// LS Electric XG5000 project: cobot_conveyor
// PLC LSPLC

PROGRAM InverterCom (task: 스캔 프로그램)

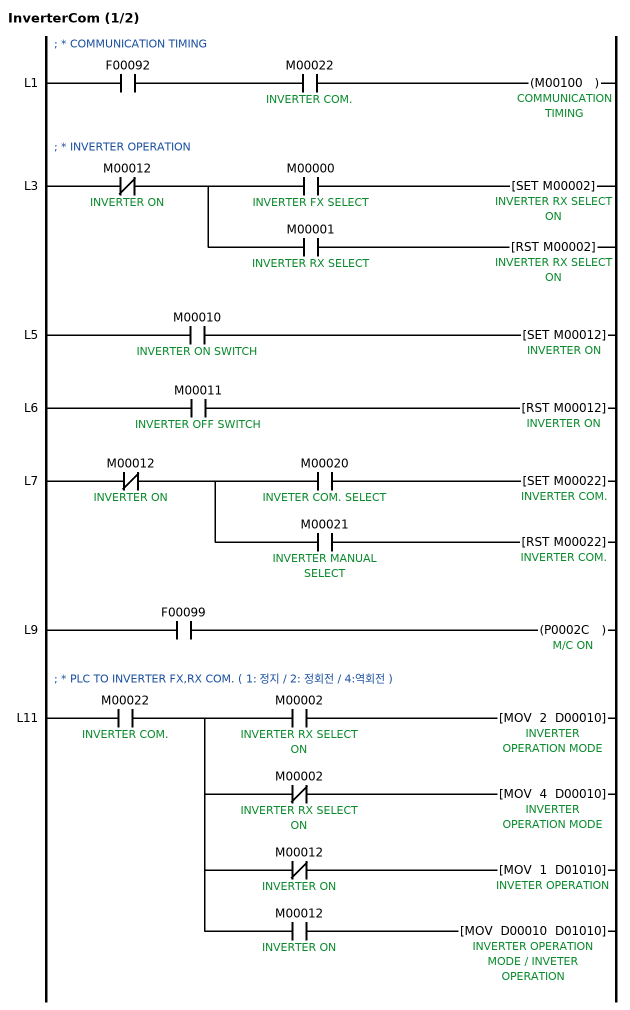
// * COMMUNICATION TIMING
; L1
LOAD      F00092
AND       M00022	// INVERTER COM.
OUT       M00100	// COMMUNICATION TIMING
// * INVERTER OPERATION
; L3
LOAD NOT  M00012	// INVERTER ON
MPUSH
AND       M00000	// INVERTER FX SELECT
SET       M00002	// INVERTER RX SELECT ON
MPOP
AND       M00001	// INVERTER RX SELECT
RST       M00002	// INVERTER RX SELECT ON
; L5
LOAD      M00010	// INVERTER ON SWITCH
SET       M00012	// INVERTER ON
; L6
LOAD      M00011	// INVERTER OFF SWITCH
RST       M00012	// INVERTER ON
; L7
LOAD NOT  M00012	// INVERTER ON
MPUSH
AND       M00020	// INVETER COM. SELECT
SET       M00022	// INVERTER COM.
MPOP
AND       M00021	// INVERTER MANUAL SELECT
RST       M00022	// INVERTER COM.
; L9
LOAD      F00099
OUT       P0002C	// M/C ON
// * PLC TO INVERTER FX,RX COM. ( 1: 정지 / 2: 정회전 / 4:역회전 )
; L11
LOAD      M00022	// INVERTER COM.
MPUSH
AND       M00002	// INVERTER RX SELECT ON
MOV       2 D00010	// INVERTER OPERATION MODE
MLOAD
AND NOT   M00002	// INVERTER RX SELECT ON
MOV       4 D00010	// INVERTER OPERATION MODE
MLOAD
AND NOT   M00012	// INVERTER ON
MOV       1 D01010	// INVETER OPERATION
MPOP
AND       M00012	// INVERTER ON
MOV       D00010 D01010	// INVERTER OPERATION MODE / INVETER OPERATION

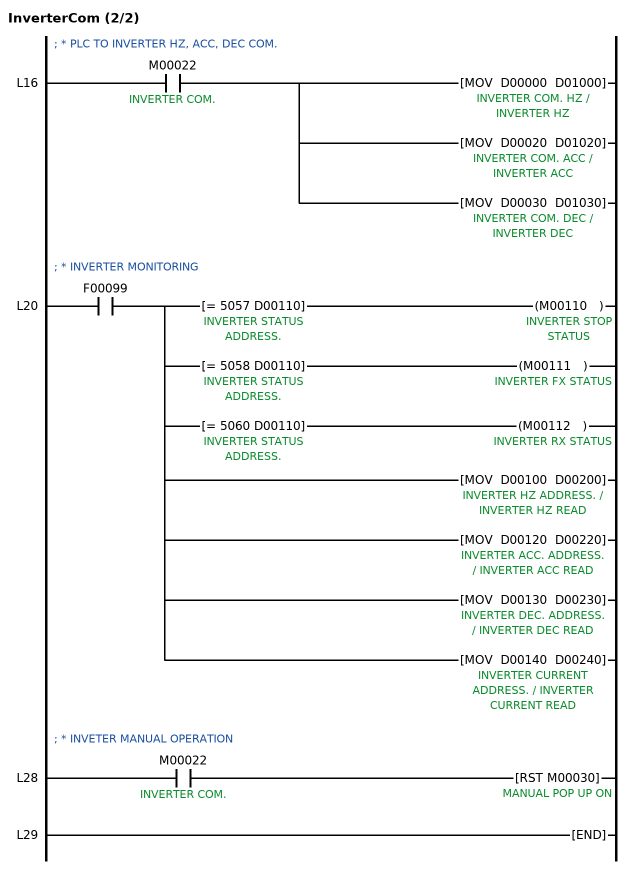
// * PLC TO INVERTER HZ, ACC, DEC COM.
; L16
LOAD      M00022	// INVERTER COM.
MOV       D00000 D01000	// INVERTER COM. HZ / INVERTER HZ
MOV       D00020 D01020	// INVERTER COM. ACC / INVERTER ACC
MOV       D00030 D01030	// INVERTER COM. DEC / INVERTER DEC
// * INVERTER MONITORING
; L20
LOAD      F00099
MPUSH
AND=      5057 D00110	// INVERTER STATUS ADDRESS.
OUT       M00110	// INVERTER STOP STATUS
MLOAD
AND=      5058 D00110	// INVERTER STATUS ADDRESS.
OUT       M00111	// INVERTER FX STATUS
MLOAD
AND=      5060 D00110	// INVERTER STATUS ADDRESS.
OUT       M00112	// INVERTER RX STATUS
MPOP
MOV       D00100 D00200	// INVERTER HZ ADDRESS. / INVERTER HZ READ
MOV       D00120 D00220	// INVERTER ACC. ADDRESS. / INVERTER ACC READ
MOV       D00130 D00230	// INVERTER DEC. ADDRESS. / INVERTER DEC READ
MOV       D00140 D00240	// INVERTER CURRENT ADDRESS. / INVERTER CURRENT READ
// * INVETER MANUAL OPERATION
; L28
LOAD      M00022	// INVERTER COM.
RST       M00030	// MANUAL POP UP ON
; L29
END

PROGRAM CountTimer (task: 스캔 프로그램)

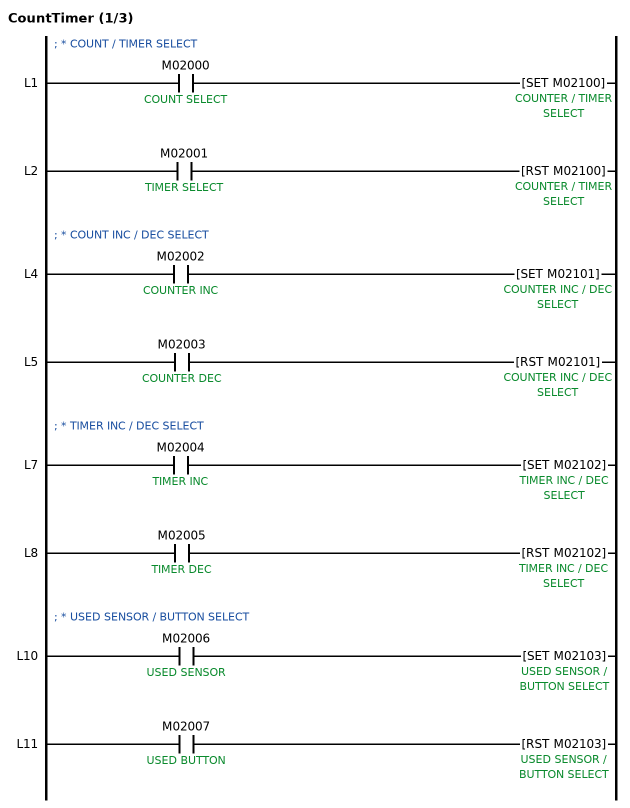
// * COUNT / TIMER SELECT
; L1
LOAD      M02000	// COUNT SELECT
SET       M02100	// COUNTER / TIMER SELECT
; L2
LOAD      M02001	// TIMER SELECT
RST       M02100	// COUNTER / TIMER SELECT
// * COUNT INC / DEC SELECT
; L4
LOAD      M02002	// COUNTER INC
SET       M02101	// COUNTER INC / DEC SELECT
; L5
LOAD      M02003	// COUNTER DEC
RST       M02101	// COUNTER INC / DEC SELECT
// * TIMER INC / DEC SELECT
; L7
LOAD      M02004	// TIMER INC
SET       M02102	// TIMER INC / DEC SELECT
; L8
LOAD      M02005	// TIMER DEC
RST       M02102	// TIMER INC / DEC SELECT
// * USED SENSOR / BUTTON SELECT
; L10
LOAD      M02006	// USED SENSOR
SET       M02103	// USED SENSOR / BUTTON SELECT
; L11
LOAD      M02007	// USED BUTTON
RST       M02103	// USED SENSOR / BUTTON SELECT

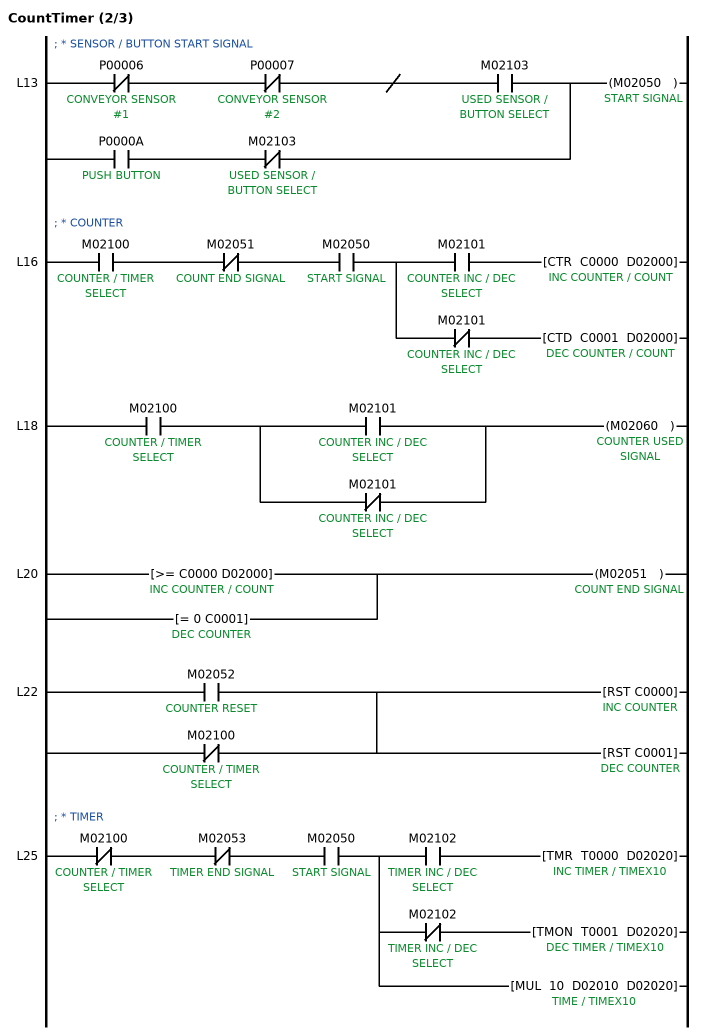
// * SENSOR / BUTTON START SIGNAL
; L13
LOAD NOT  P00006	// CONVEYOR SENSOR #1
AND NOT   P00007	// CONVEYOR SENSOR #2
NOT
AND       M02103	// USED SENSOR / BUTTON SELECT
LOAD      P0000A	// PUSH BUTTON
AND NOT   M02103	// USED SENSOR / BUTTON SELECT
OR LOAD
OUT       M02050	// START SIGNAL
// * COUNTER
; L16
LOAD      M02100	// COUNTER / TIMER SELECT
AND NOT   M02051	// COUNT END SIGNAL
AND       M02050	// START SIGNAL
MPUSH
AND       M02101	// COUNTER INC / DEC SELECT
CTR       C0000 D02000	// INC COUNTER / COUNT
MPOP
AND NOT   M02101	// COUNTER INC / DEC SELECT
CTD       C0001 D02000	// DEC COUNTER / COUNT
; L18
LOAD      M02100	// COUNTER / TIMER SELECT
LOAD      M02101	// COUNTER INC / DEC SELECT
OR NOT    M02101	// COUNTER INC / DEC SELECT
AND LOAD
OUT       M02060	// COUNTER USED SIGNAL
; L20
LOAD>=    C0000 D02000	// INC COUNTER / COUNT
OR=       0 C0001	// DEC COUNTER
OUT       M02051	// COUNT END SIGNAL
; L22
LOAD      M02052	// COUNTER RESET
OR NOT    M02100	// COUNTER / TIMER SELECT
RST       C0000	// INC COUNTER
RST       C0001	// DEC COUNTER
// * TIMER
; L25
LOAD NOT  M02100	// COUNTER / TIMER SELECT
AND NOT   M02053	// TIMER END SIGNAL
AND       M02050	// START SIGNAL
MPUSH
AND       M02102	// TIMER INC / DEC SELECT
TMR       T0000 D02020	// INC TIMER / TIMEX10
MLOAD
AND NOT   M02102	// TIMER INC / DEC SELECT
TMON      T0001 D02020	// DEC TIMER / TIMEX10
MPOP
MUL       10 D02010 D02020	// TIME / TIMEX10

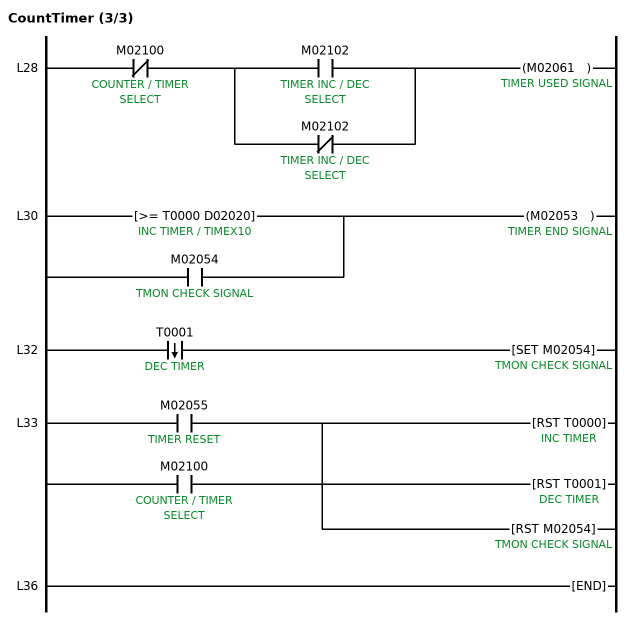
; L28
LOAD NOT  M02100	// COUNTER / TIMER SELECT
LOAD      M02102	// TIMER INC / DEC SELECT
OR NOT    M02102	// TIMER INC / DEC SELECT
AND LOAD
OUT       M02061	// TIMER USED SIGNAL
; L30
LOAD>=    T0000 D02020	// INC TIMER / TIMEX10
OR        M02054	// TMON CHECK SIGNAL
OUT       M02053	// TIMER END SIGNAL
; L32
LOADN     T0001	// DEC TIMER
SET       M02054	// TMON CHECK SIGNAL
; L33
LOAD      M02055	// TIMER RESET
OR        M02100	// COUNTER / TIMER SELECT
RST       T0000	// INC TIMER
RST       T0001	// DEC TIMER
RST       M02054	// TMON CHECK SIGNAL
; L36
END

PROGRAM Button (task: 스캔 프로그램)

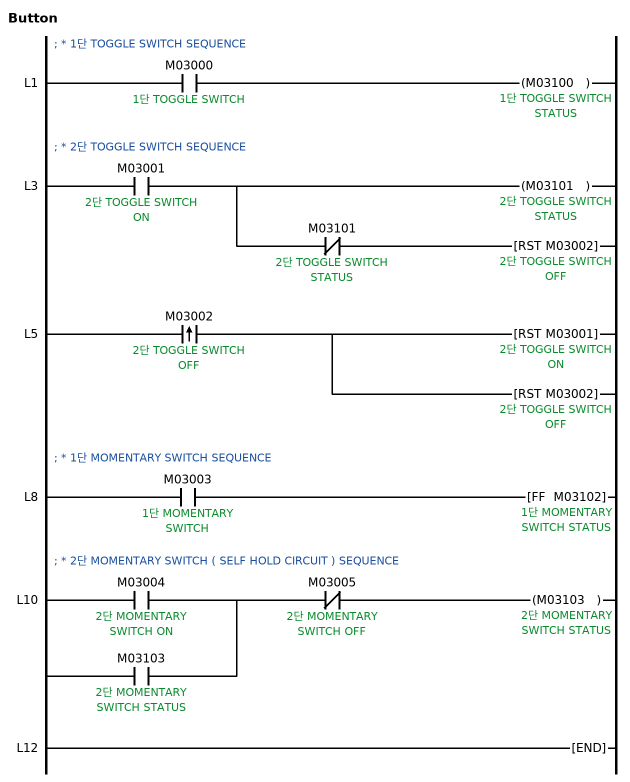
// * 1단 TOGGLE SWITCH SEQUENCE
; L1
LOAD      M03000	// 1단 TOGGLE SWITCH
OUT       M03100	// 1단 TOGGLE SWITCH STATUS
// * 2단 TOGGLE SWITCH SEQUENCE
; L3
LOAD      M03001	// 2단 TOGGLE SWITCH ON
OUT       M03101	// 2단 TOGGLE SWITCH STATUS
AND NOT   M03101	// 2단 TOGGLE SWITCH STATUS
RST       M03002	// 2단 TOGGLE SWITCH OFF
; L5
LOADP     M03002	// 2단 TOGGLE SWITCH OFF
RST       M03001	// 2단 TOGGLE SWITCH ON
RST       M03002	// 2단 TOGGLE SWITCH OFF
// * 1단 MOMENTARY SWITCH SEQUENCE
; L8
LOAD      M03003	// 1단 MOMENTARY SWITCH
FF        M03102	// 1단 MOMENTARY SWITCH STATUS
// * 2단 MOMENTARY SWITCH ( SELF HOLD CIRCUIT ) SEQUENCE
; L10
LOAD      M03004	// 2단 MOMENTARY SWITCH ON
OR        M03103	// 2단 MOMENTARY SWITCH STATUS
AND NOT   M03005	// 2단 MOMENTARY SWITCH OFF
OUT       M03103	// 2단 MOMENTARY SWITCH STATUS
; L12
END

PROGRAM Manual (task: 스캔 프로그램)

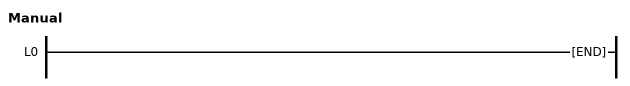
; L0
END

PROGRAM Button_control (task: 스캔 프로그램)

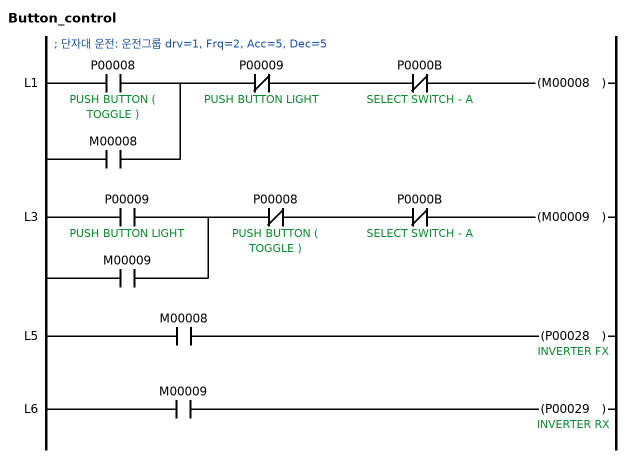
// 단자대 운전: 운전그룹 drv=1, Frq=2, Acc=5, Dec=5
; L1
LOAD      P00008	// PUSH BUTTON ( TOGGLE )
OR        M00008
AND NOT   P00009	// PUSH BUTTON LIGHT
AND NOT   P0000B	// SELECT SWITCH - A
OUT       M00008
; L3
LOAD      P00009	// PUSH BUTTON LIGHT
OR        M00009
AND NOT   P00008	// PUSH BUTTON ( TOGGLE )
AND NOT   P0000B	// SELECT SWITCH - A
OUT       M00009
; L5
LOAD      M00008
OUT       P00028	// INVERTER FX
; L6
LOAD      M00009
OUT       P00029	// INVERTER RX

PROGRAM control (task: 스캔 프로그램)

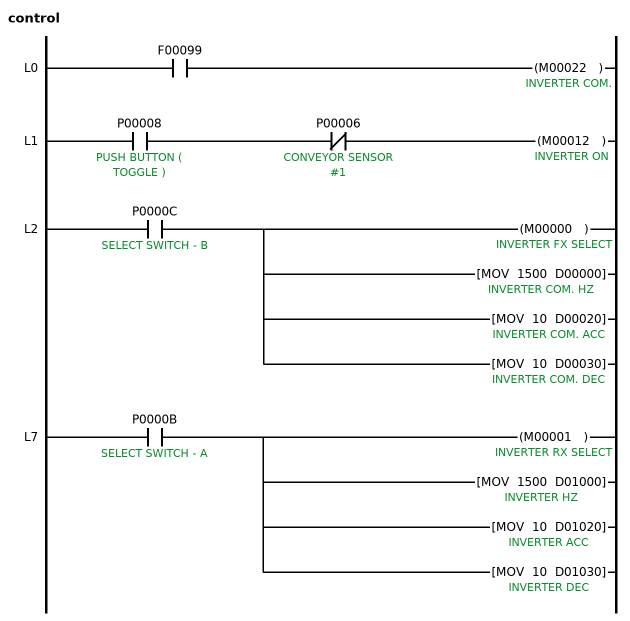
; L0
LOAD      F00099
OUT       M00022	// INVERTER COM.
; L1
LOAD      P00008	// PUSH BUTTON ( TOGGLE )
AND NOT   P00006	// CONVEYOR SENSOR #1
OUT       M00012	// INVERTER ON
; L2
LOAD      P0000C	// SELECT SWITCH - B
OUT       M00000	// INVERTER FX SELECT
MOV       1500 D00000	// INVERTER COM. HZ
MOV       10 D00020	// INVERTER COM. ACC
MOV       10 D00030	// INVERTER COM. DEC
; L7
LOAD      P0000B	// SELECT SWITCH - A
OUT       M00001	// INVERTER RX SELECT
MOV       1500 D01000	// INVERTER HZ
MOV       10 D01020	// INVERTER ACC
MOV       10 D01030	// INVERTER DEC

VARIABLES AND COMMENTS (devices not used above)
P00000	BIT	COUNTER / TIMER OUTPUT
P00001	BIT	INVERTER OUTPUT
P00002	BIT	M/S ON STATUS
P00020	BIT	COUNT PULSE
P00021	BIT	TIMER HOLD
P00022	BIT	RESET
P00024	BIT	RED LAMP ON
P00025	BIT	YELLOW LAMP ON
P00026	BIT	GREEN LAMP ON